FUNCTION_BLOCK FB_TrackBase
VAR_INPUT
END_VAR
VAR_OUTPUT
	bBusy 	: BOOL;
	bError 	: BOOL;
END_VAR
VAR
	trackLinePosStart 	: PositionXYC;
	trackLinePosEnd 	: PositionXYC;
	fbTrackStandard		: FB_TrackStandard;
	fTrackLength		: LREAL;
END_VAR

METHOD ccl00_cycle : BOOL
VAR_INPUT
END_VAR
fbTrackStandard.Cycle();
END_METHOD

PROPERTY P_TrackLength : LREAL
GET
P_TrackLength := fTrackLength;
END_GET
END_PROPERTY

PROPERTY std : I_TrackStandard
GET
std := fbTrackStandard;
END_GET
END_PROPERTY

END_FUNCTION_BLOCK

(* stored: Version 1.1.0.1, ProductVersion 3.1.4024.9
   POU FB_TrackBase: Id {c3c3f9fa-5ce3-4074-9364-756b12d0b77f}, SpecialFunc None
   Method ccl00_cycle: Id {fdee6f85-73f9-4381-bd15-490efb065389}
   Property P_TrackLength: Id {de37312d-e30d-4920-ad38-7645514e566b}
   Get Get: Id {b776e306-77dd-4def-b958-9f6aa2dc687d}
   Property std: Id {9be86626-2dbf-44cd-9915-089d605f0a97}
   Get Get: Id {895572ff-f985-4450-b868-37aab89a00b8} *)
